# EPICS autosave request: trunk/stdApp/Db/genericStrState_settings.req
$(P)$(S)val$(N).VAL
$(P)$(S)mode$(N).VAL
$(P)$(S)pv$(N).VAL
